Fanuc KAREL source: ka00122.KL

-- PROVISIONAL review KL for V1013-1; original PC SHA256 aae8508434fe66e7f8a0987ce641c7976b782d2956b4db5ba19b45ac4c2e279b
-- Incomplete behavior may be omitted. Consult companion uncertainty JSON. Do not deploy.
PROGRAM KA00122
%NOLOCKGROUP
VAR
  DST : REAL
-- UNRESOLVED_DECL SRC type=002018
BEGIN
  -- UNRESOLVED_PC offsets 5-19; opcodes 2E,22,9D,33,B2
  -- UNRESOLVED_PC offsets 24-40; opcodes 22,9D,33,B1,64,23
  -- UNRESOLVED_PC offsets 45-49; opcodes 7F
END KA00122
